FUNCTION F_UpdateParametersByReference_1 
VAR_INPUT
	bSetNewValue : BOOL;
	fMaxPistonStroke : LREAL;
	paramCylinderPiston : REFERENCE TO ST_PistonRange;
END_VAR
VAR

END_VAR

IF bSetNewValue THEN
	paramCylinderPiston.fPistonPosMax := fMaxPistonStroke;
	bSetNewValue := FALSE;
END_IF

END_FUNCTION

(* stored: Version 1.1.0.1, ProductVersion 3.1.4024.10
   POU F_UpdateParametersByReference_1: Id {99761e76-756a-496d-9e5c-a61054bb3a02}, SpecialFunc None *)
